FUNCTION_BLOCK FB_Event EXTENDS FB_ListString IMPLEMENTS I_Event
VAR_INPUT
	bExecute:   		BOOL;
	fbObserver:			FB_Observer;
END_VAR
VAR_OUTPUT
END_VAR
VAR
	iParent:			I_Component;
	stError:			ST_Event;
END_VAR

SUPER^();
fbObserver();

METHOD FB_init : BOOL
VAR_INPUT
	bInitRetains : BOOL; // if TRUE, the retain variables are initialized (warm start / cold start)
	bInCopyCode : BOOL;  // if TRUE, the instance afterwards gets moved into the copy code (online change)
	iParent:			I_Component;
END_VAR
THIS^.iParent:= iParent;
END_METHOD

METHOD PUBLIC M_Abort : BOOL
VAR_INPUT
	Message:				STRING(255);
	ID:						UDINT;
END_VAR

stError.Timestamp:= F_GetSystemTime();
stError.Message:= Message;
stError.ID:= ID;
stError.Arguments:= M_Arguments();

iParent.M_Request(E_Request.Abort);
fbObserver.M_Notify(E_Request.Abort);
M_Clear();
END_METHOD

METHOD INTERNAL M_Arguments : STRING(255)
VAR_INPUT
END_VAR
VAR
	nIndex:			INT;
END_VAR
WHILE nIndex < nLength DO
	M_Arguments:= Concat(Concat(M_Arguments, pList[nIndex]), '$N');
	nIndex:= nIndex + 1;
END_WHILE
END_METHOD

METHOD PUBLIC M_Debug : BOOL
VAR_INPUT
	Message:				STRING(255);
END_VAR
END_METHOD

METHOD PUBLIC M_Error : BOOL
VAR_INPUT
	Message:				STRING(255);
	ID:						UDINT;
END_VAR

stError.Timestamp:= F_GetSystemTime();
stError.Message:= Message;
stError.ID:= ID;
stError.Arguments:= M_Arguments();

fbObserver.M_Notify(E_State.Aborted);
M_Clear();
END_METHOD

METHOD PUBLIC M_Information : BOOL
VAR_INPUT
	Message:				STRING(255);
	ID:						UDINT;
END_VAR
END_METHOD

METHOD PUBLIC M_Stop : BOOL
VAR_INPUT
	Message:				STRING(255);
	ID:						UDINT;
END_VAR

stError.Timestamp:= F_GetSystemTime();
stError.Message:= Message;
stError.ID:= ID;
stError.Arguments:= M_Arguments();

iParent.M_Request(E_Request.Stop);
fbObserver.M_Notify(E_Request.Stop);
M_Clear();
END_METHOD

METHOD PUBLIC M_Warning : BOOL
VAR_INPUT
	Message:				STRING(255);
	ID:						UDINT;
END_VAR
END_METHOD

PROPERTY PUBLIC P_Observer : I_Observer
GET
P_Observer:= fbObserver;
END_GET
END_PROPERTY

END_FUNCTION_BLOCK

(* stored: Version 1.1.0.1
   POU FB_Event: Id {59616103-7f2e-4b6f-81bd-583969a36d28}, SpecialFunc None
   Method FB_init: Id {be23ffcc-529d-4010-ace3-b17baed191a5}
   Method M_Abort: Id {55348828-4763-4c06-9dd1-090fa29a8379}
   Method M_Arguments: Id {70779266-7b36-4bce-9e6f-049e951fd75a}
   Method M_Debug: Id {0a2b992b-2a4a-0251-0210-713b326debf6}
   Method M_Error: Id {dedc6a92-4fd3-0050-1590-6a55ab6d568e}
   Method M_Information: Id {d9a244f2-1d6f-434f-aab4-cad6aacbb94f}
   Method M_Stop: Id {089fbf49-839d-443a-b3f2-2540679d46a9}
   Method M_Warning: Id {d443b8bb-774e-487e-80a2-79cf66a0376c}
   Property P_Observer: Id {2b4a3b9d-02d6-46ef-a830-8f731a2ada59}
   Get Get: Id {d2313d10-2a66-4a0c-9a20-b577c055dab4} *)
